INTERFACE ITF_Configuration

METHOD PUBLIC AddTopElementToLogger : BOOL
VAR_INPUT
END_VAR
END_METHOD

(*			
	RafalOS
	Rafał Osajda		29.10.2025		TC 4024.66
	Dodawanie TopElementu do systemu
*)
METHOD PUBLIC AddTopElementToMachineControl : BOOL
VAR_INPUT
	itfMachineControl			: ITF_MachineControlConfigure;
END_VAR
END_METHOD

METHOD PUBLIC SetStartMode : BOOL
VAR_INPUT
	itfMachineControl			: ITF_MachineControlConfigure;
END_VAR
END_METHOD

METHOD StateAndModes : BOOL
VAR_INPUT
	itfMachineControl			: ITF_MachineControlConfigure;
END_VAR
END_METHOD

END_INTERFACE

(* stored: Version 1.1.0.1
   Itf ITF_Configuration: Id {687dfd14-96fc-4e9e-9986-638f15f5b1fd}
   Method AddTopElementToLogger: Id {a4cd0c5f-7f5c-0a74-2586-ca395c8c0f41}
   Method AddTopElementToMachineControl: Id {8b896f22-6be0-0e79-09a1-eb54c9dc66d6}
   Method SetStartMode: Id {36444d97-b5e1-0e95-31fa-e113c6730599}
   Method StateAndModes: Id {58f0fcc3-ac6f-0f4f-040a-f5ab763b7603} *)
